FUNCTION_BLOCK differential_protection_1_3 (* Composite Function Block Type *)
  (* Standard: 61499-2 *)
  (* Version 0.0, 3/23/2016, gulzha, nxtControl GmbH, template *)
  PACKAGE Main;
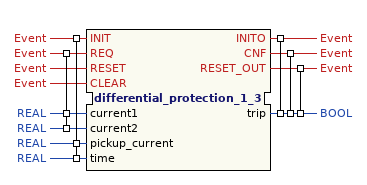
  EVENT_INPUT
    INIT WITH pickup_current, time; (* Initialization Request *)
    REQ WITH current1, current2; (* Normal Execution Request *)
    RESET;
    CLEAR;
  END_EVENT
  EVENT_OUTPUT
    INITO WITH trip; (* Initialization Confirm *)
    CNF WITH trip; (* Execution Confirmation *)
    RESET_OUT WITH trip;
  END_EVENT
  VAR_INPUT
    current1 : REAL;
    current2 : REAL;
    pickup_current : REAL;
    time : REAL;
  END_VAR
  VAR_OUTPUT
    trip : BOOL;
  END_VAR
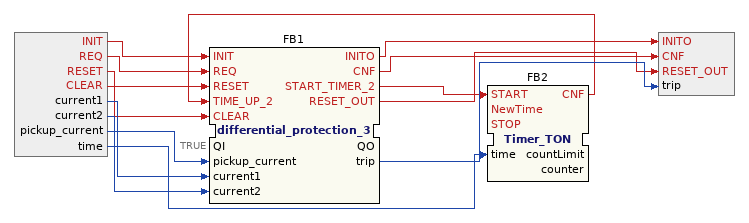
  FBS
    FB1 : differential_protection_3(QI := TRUE);
    FB2 : Timer_TON;
  END_FBS
  EVENT_CONNECTIONS
    INIT TO FB1.INIT;
    FB1.INITO TO INITO;
    FB1.CNF TO CNF;
    REQ TO FB1.REQ;
    RESET TO FB1.RESET;
    FB1.RESET_OUT TO RESET_OUT;
    CLEAR TO FB1.CLEAR;
    FB1.START_TIMER_2 TO FB2.START;
    FB2.CNF TO FB1.TIME_UP_2;
  END_CONNECTIONS
  DATA_CONNECTIONS
    FB1.trip TO trip;
    pickup_current TO FB1.pickup_current;
    current1 TO FB1.current1;
    current2 TO FB1.current2;
    time TO FB2.time;
  END_CONNECTIONS
END_FUNCTION_BLOCK
